INTERFACE ITF_Button EXTENDS ITF_BaseComponent

METHOD PUBLIC GetRisingEdgePressed : BOOL
VAR_INPUT
END_VAR
END_METHOD

(*			
	EVERDE sp. z o.o.
	Rafał Osajda		31.01.2025		TC 4026.13		wer. 0.0.0.1
	Zwraca stan przycisku
*)
METHOD IsPressed : BOOL
END_METHOD

END_INTERFACE

(* stored: Version 1.1.0.1
   Itf ITF_Button: Id {16024c1d-6861-43f4-a8ee-1b1c23148973}
   Method GetRisingEdgePressed: Id {623d085c-062a-0c39-3d2b-a7efe6ed305a}
   Method IsPressed: Id {92495ad2-c596-475f-8486-e61a1b02cd06} *)
